FUNCTION F_GetErrorId : UDINT;
VAR_INPUT
	Feedback : I_CommandFeedback;
END_VAR

IF Feedback <> 0 THEN
	F_GetErrorId := Feedback.ErrorId;
END_IF

END_FUNCTION

(* stored: Version 1.1.0.1, ProductVersion 3.1.4024.12
   POU F_GetErrorId: Id {4ac7a0ff-10d3-07d0-0e2f-05a1a934aee0}, SpecialFunc None *)
